FUNCTION_BLOCK GaitPlanner
VAR_INPUT
END_VAR
VAR_OUTPUT
END_VAR
VAR
	gaitCount : UDINT := 0;
	recoverGaitPlanner : RecoverGait;
	StaticwalkGaitPlanner    : StaticWalkGait;
	liftBodyGaitPlanner    : LiftBodyGait;
	swingBodyGaitPlanner : SwingBodyGait;
	CurlingGaitPlanner :CurlingGait;
	CurlingGaitPlanner2 :CurlingGaitFromStance;
	RcToSlipFromCurlingPlanner:RcToSlipFromCurling;
	BLegSlipPlanner:BLegSlip;
	CurlingGaitFromSlipPlanner:CurlingGaitFromSlip;
	RcToCurlingFromSlipPlanner:RcToCurlingFromSlip;
	RcToStanceFromSlipPlanner:RcToStanceFromSlip;
	TrotWalkPlanner:TrotWalk;
	WalkSlopePlanner : WalkSlopeGait;
	
	
END_VAR

METHOD PUBLIC DoPlanning : BOOL
VAR_INPUT
END_VAR
VAR_OUTPUT
	isDone : BOOL;
END_VAR

VAR
	i: INT;
	j: INT;
END_VAR
IF gvl.gaitId = 0 THEN
	recoverGaitPlanner.DoPlanning(gaitCount);
	isDone := recoverGaitPlanner.isFinished;
	FOR i := 0 TO 5 DO
		FOR j := 0 TO 2 DO
			gvl.jntRefPosTuning[i, j] := recoverGaitPlanner.jointPosTarget[i, j];
			gvl.jntRefVelTuning[i, j] := recoverGaitPlanner.jointVelTarget[i, j];
			gvl.jntRefFceTuning[i, j] := recoverGaitPlanner.jointFceTarget[i, j];
		END_FOR
	END_FOR
ELSIF gvl.gaitId = 1 THEN
	StaticwalkGaitPlanner.DoPlanning(gaitCount);
	isDone := StaticwalkGaitPlanner.isFinished;
	FOR i := 0 TO 5 DO
		FOR j := 0 TO 2 DO
			gvl.jntRefPosTuning[i, j] := StaticwalkGaitPlanner.jointPosTarget[i, j];
			gvl.jntRefVelTuning[i, j] := StaticwalkGaitPlanner.jointVelTarget[i, j];
			gvl.jntRefFceTuning[i, j] := StaticwalkGaitPlanner.jointFceTarget[i, j];
		END_FOR
	END_FOR
ELSIF gvl.gaitId = 2 THEN
	liftBodyGaitPlanner.DoPlanning(count:=gaitCount );
	isDone := liftBodyGaitPlanner.isFinished;
	FOR i := 0 TO 5 DO
		FOR j := 0 TO 2 DO
			gvl.jntRefPosTuning[i, j] := liftBodyGaitPlanner.jointPosTarget[i, j];
			gvl.jntRefVelTuning[i, j] := liftBodyGaitPlanner.jointVelTarget[i, j];
			gvl.jntRefFceTuning[i, j] := liftBodyGaitPlanner.jointFceTarget[i, j];
		END_FOR
	END_FOR	

ELSIF gvl.gaitId = 3 THEN
	swingBodyGaitPlanner.DoPlanning(gaitCount);
	isDone := swingBodyGaitPlanner.isFinished;
	FOR i := 0 TO 5 DO
		FOR j := 0 TO 2 DO
			gvl.jntRefPosTuning[i, j] := swingBodyGaitPlanner.jointPosTarget[i, j];
			gvl.jntRefVelTuning[i, j] := swingBodyGaitPlanner.jointVelTarget[i, j];
			gvl.jntRefFceTuning[i, j] := swingBodyGaitPlanner.jointFceTarget[i, j];
		END_FOR
	END_FOR
ELSIF gvl.gaitId = 4 THEN
	CurlingGaitPlanner2.DoPlanning(gaitCount);
	isDone := CurlingGaitPlanner2.isFinished;
	FOR i := 0 TO 5 DO
		FOR j := 0 TO 2 DO
			gvl.jntRefPosTuning[i, j] := CurlingGaitPlanner2.jointPosTarget[i, j];
			gvl.jntRefVelTuning[i, j] := CurlingGaitPlanner2.jointVelTarget[i, j];
			gvl.jntRefFceTuning[i, j] := CurlingGaitPlanner2.jointFceTarget[i, j];
		END_FOR
	END_FOR
ELSIF gvl.gaitId = 5 THEN
	CurlingGaitFromSlipPlanner.DoPlanning(gaitCount);
	isDone := CurlingGaitFromSlipPlanner.isFinished;
	FOR i := 0 TO 5 DO
		FOR j := 0 TO 2 DO
			gvl.jntRefPosTuning[i, j] := CurlingGaitFromSlipPlanner.jointPosTarget[i, j];
			gvl.jntRefVelTuning[i, j] := CurlingGaitFromSlipPlanner.jointVelTarget[i, j];
			gvl.jntRefFceTuning[i, j] := CurlingGaitFromSlipPlanner.jointFceTarget[i, j];
		END_FOR
	END_FOR
ELSIF gvl.gaitId = 6 THEN
	RcToSlipFromCurlingPlanner.DoPlanning(gaitCount);
	isDone := RcToSlipFromCurlingPlanner.isFinished;
	FOR i := 0 TO 5 DO
		FOR j := 0 TO 2 DO
			gvl.jntRefPosTuning[i, j] := RcToSlipFromCurlingPlanner.jointPosTarget[i, j];
			gvl.jntRefVelTuning[i, j] := RcToSlipFromCurlingPlanner.jointVelTarget[i, j];
			gvl.jntRefFceTuning[i, j] := RcToSlipFromCurlingPlanner.jointFceTarget[i, j];
		END_FOR
	END_FOR
ELSIF gvl.gaitId = 7 THEN
	RcToCurlingFromSlipPlanner.DoPlanning(gaitCount);
	isDone := RcToCurlingFromSlipPlanner.isFinished;
	FOR i := 0 TO 5 DO
		FOR j := 0 TO 2 DO
			gvl.jntRefPosTuning[i, j] := RcToCurlingFromSlipPlanner.jointPosTarget[i, j];
			gvl.jntRefVelTuning[i, j] := RcToCurlingFromSlipPlanner.jointVelTarget[i, j];
			gvl.jntRefFceTuning[i, j] := RcToCurlingFromSlipPlanner.jointFceTarget[i, j];
		END_FOR
	END_FOR
ELSIF gvl.gaitId = 8 THEN
	RcToStanceFromSlipPlanner.DoPlanning(gaitCount);
	isDone := RcToStanceFromSlipPlanner.isFinished;
	FOR i := 0 TO 5 DO
		FOR j := 0 TO 2 DO
			gvl.jntRefPosTuning[i, j] := RcToStanceFromSlipPlanner.jointPosTarget[i, j];
			gvl.jntRefVelTuning[i, j] := RcToStanceFromSlipPlanner.jointVelTarget[i, j];
			gvl.jntRefFceTuning[i, j] := RcToStanceFromSlipPlanner.jointFceTarget[i, j];
		END_FOR
	END_FOR
ELSIF gvl.gaitId = 9 THEN
	BLegSlipPlanner.DoPlanning(gaitCount);
	isDone := BLegSlipPlanner.isFinished;
	FOR i := 0 TO 5 DO
		FOR j := 0 TO 2 DO
			gvl.jntRefPosTuning[i, j] := BLegSlipPlanner.jointPosTarget[i, j];
			gvl.jntRefVelTuning[i, j] := BLegSlipPlanner.jointVelTarget[i, j];
			gvl.jntRefFceTuning[i, j] := BLegSlipPlanner.jointFceTarget[i, j];
		END_FOR
	END_FOR
ELSIF gvl.gaitId = 10 THEN
	TrotWalkPlanner.DoPlanning(gaitCount);
	isDone := TrotWalkPlanner.isFinished;
	FOR i := 0 TO 5 DO
		FOR j := 0 TO 2 DO
			gvl.jntRefPosTuning[i, j] := TrotWalkPlanner.jointPosTarget[i, j];
			gvl.jntRefVelTuning[i, j] := TrotWalkPlanner.jointVelTarget[i, j];
			gvl.jntRefFceTuning[i, j] := TrotWalkPlanner.jointFceTarget[i, j];
		END_FOR
	END_FOR
ELSIF gvl.gaitId = 11 THEN
	WalkSlopePlanner.DoPlanning(gaitCount);
	isDone := WalkSlopePlanner.isFinished;
	FOR i := 0 TO 5 DO
		FOR j := 0 TO 2 DO
			gvl.jntRefPosTuning[i, j] := WalkSlopePlanner.jointPosTarget[i, j];
			gvl.jntRefVelTuning[i, j] := WalkSlopePlanner.jointVelTarget[i, j];
			gvl.jntRefFceTuning[i, j] := WalkSlopePlanner.jointFceTarget[i, j];
		END_FOR
	END_FOR
ELSE
	// no gait selected
	FOR i := 0 TO 5 DO
		FOR j := 0 TO 2 DO
			IF ABS(gvl.jntActualPos[i, j]-gvl.lastjntRefPos[i,j])<0.1 THEN
				gvl.jntRefPosTuning[i, j] :=gvl.lastjntRefPos[i,j];
			ELSE
				gvl.jntRefPosTuning[i, j] := gvl.jntActualPos[i, j];				
			END_IF
			gvl.jntRefVelTuning[i, j] := 0;
			gvl.jntRefFceTuning[i, j] := 0;
		END_FOR
	END_FOR
	isDone := TRUE;
END_IF

//Tuning state 
(*FOR i := 0 TO 5 DO
	FOR j := 0 TO 2 DO
			IF ABS(gvl.jntActualPos[i, j]-gvl.lastjntRefPos[i,j])<0.1 THEN
				gvl.jntRefPos[i, j] :=gvl.lastjntRefPos[i,j];
			ELSE
				gvl.jntRefPos[i, j] := gvl.jntActualPos[i, j];				
			END_IF
		gvl.jntRefVel[i, j] := 0;
		gvl.jntRefFce[i, j] := 0;
	END_FOR
END_FOR*)

//Actual employment
gvl.jntRefPos:=gvl.jntRefPosTuning;
gvl.jntRefVel:=gvl.jntRefVelTuning;
gvl.jntRefFce:=gvl.jntRefFceTuning;

gaitCount := gaitCount + 1;
END_METHOD

METHOD PUBLIC FinalizeGaitCmd : BOOL
VAR_INPUT
END_VAR

VAR
	i: INT;
	j: INT;
END_VAR
FOR i := 0 TO 5 DO
	FOR j := 0 TO 2 DO
		//gvl.jntRefPos[i, j] := gvl.jntActualPos[i, j];
		gvl.jntRefVel[i, j] := 0;
		gvl.jntRefFce[i, j] := 0;
	END_FOR
END_FOR
END_METHOD

METHOD PUBLIC Initialize : BOOL
VAR_INPUT
END_VAR
gaitCount := 0;
END_METHOD

END_FUNCTION_BLOCK

(* stored: Version 1.1.0.1, ProductVersion 3.1.4024.2
   POU GaitPlanner: Id {e28e8e20-85b5-4fe0-bcf3-a17b16517cf7}, SpecialFunc None
   Method DoPlanning: Id {b671005c-502a-4e79-9952-da78632d7259}
   Method FinalizeGaitCmd: Id {1655f237-6311-4aea-bffb-4de8aa2fd652}
   Method Initialize: Id {c1c79418-21b5-4a6b-bb9b-d3a40ca6d8bc} *)
